(* IEC 61131-3 sources: AutomationLab/ConveyerObject/Model, 3 files *)

(* ---- Conveyer.st ---- *)
FUNCTION_BLOCK Conveyer
VAR_INPUT
END_VAR
VAR_OUTPUT
END_VAR
VAR
END_VAR
VAR_IN_OUT
	Data: ConveyerType;
END_VAR

Data.ComRotateLent := AlwaysOn(Allow:= NOT Data.BoxOnEndPosition);

(* ---- Conveyer1.st ---- *)
// ============================================
// ФУНКЦИОНАЛЬНЫЙ БЛОК — управление конвейером
// ============================================
FUNCTION_BLOCK Conveyer1
VAR_INPUT
    SensorA: BOOL; // Сигнал с датчика
END_VAR
VAR_OUTPUT
    RotateLent: BOOL; // Команда вращения ленты
END_VAR
VAR
    DelayTon: TON; // таймер задержки срабатывания
    DelayTime: TIME := T#100ms; // время задержки
END_VAR

// задержка срабатывания блока
DelayTon(IN := NOT SensorA, PT := DelayTime, Q => RotateLent);

END_FUNCTION_BLOCK

(* ---- Conveyer_FB.st ---- *)
FUNCTION_BLOCK Conveyer_FB
VAR_INPUT
END_VAR
VAR_OUTPUT
END_VAR
VAR
END_VAR
VAR_IN_OUT
	Data: ConveyerType;
END_VAR

Data.ComRotateLent := NOT Data.BoxOnEndPosition;
